FUNCTION_BLOCK TurnTableControllerIProv (* Turn Table Controller Interface Provider *)
  (* Standard: 61499-2 *)
  (* Version 0.2, 2003-12-05, JHC, Rockwell Automation, Renamed from NEWCOMPFB. *)
  (* Version 0.1, 2002-01-08, JHC, Rockwell Automation, Added DLY FB as example. *)
  (* Version 0.0, 2000-05-27, JHC, Rockwell Automation *)
  (* Compiler header: package fb.rt.dasdA1.A2.TurnTable; *)
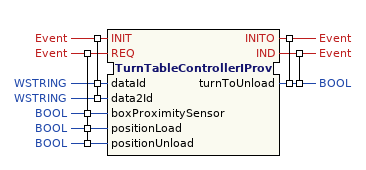
  EVENT_INPUT
    INIT WITH dataId, data2Id; (* Initialization Request *)
    REQ WITH boxProximitySensor, positionLoad, positionUnload;
  END_EVENT
  EVENT_OUTPUT
    INITO WITH turnToUnload; (* Initialization Confirm *)
    IND WITH turnToUnload;
  END_EVENT
  VAR_INPUT
    dataId : WSTRING;
    data2Id : WSTRING;
    boxProximitySensor : BOOL;
    positionLoad : BOOL;
    positionUnload : BOOL;
  END_VAR
  VAR_OUTPUT
    turnToUnload : BOOL;
  END_VAR
  FBS
    data : SUBL_1;
    data2 : PUBL_3;
  END_FBS
  EVENT_CONNECTIONS
    INIT TO data.INIT;
    data.IND TO IND;
    data.INITO TO data2.INIT;
    REQ TO data2.REQ;
    data2.INITO TO INITO;
  END_CONNECTIONS
  DATA_CONNECTIONS
    dataId TO data.ID;
    data.RD_1 TO turnToUnload;
    data2Id TO data2.ID;
    boxProximitySensor TO data2.SD_1;
    positionLoad TO data2.SD_2;
    positionUnload TO data2.SD_3;
  END_CONNECTIONS
END_FUNCTION_BLOCK
